FUNCTION_BLOCK fbUN
VAR_IN_OUT
	un : ST_UN;
	cell : ST_CELL;
END_VAR

VAR_INPUT
	EnableSim : BOOL;
END_VAR

END_FUNCTION_BLOCK

(* stored: Version 1.1.0.1, ProductVersion 3.1.4024.12
   POU fbUN: Id {ccbda342-45e8-4570-b3b5-a767274183ee}, SpecialFunc None *)
